{attribute 'qualified_only'}
VAR_GLOBAL
END_VAR

(* stored: Version 1.1.0.1, ProductVersion 3.1.4024.12
   GVL myList: Id {fadeb117-ee2b-40f9-817d-349c14b4b5bf} *)
